{attribute 'GeneratedUsingTerminal: EL3413-0000-0019'}
{attribute addProperty BoxType "EL3413-0000-0019"}
{attribute addProperty Id "PM_Inputs_Channel_1AT %I*PM_Inputs_Channel_345EAE5425PM_Inputs_Channel_2AT %I*PM_Inputs_Channel_345EAE5425PM_Inputs_Channel_3AT %I*PM_Inputs_Channel_345EAE5425PM_Inputs_AuxiliaryAT %I*PM_Inputs_Auxiliary_3661DB6D9PM_Outputs_Channel_1AT %Q*PM_Outputs_Channel_E5FBDE301PM_Outputs_Channel_2AT %Q*PM_Outputs_Channel_E5FBDE301PM_Outputs_Channel_3AT %Q*PM_Outputs_Channel_E5FBDE301PM_Outputs_AuxiliaryAT %Q*PM_Outputs_Auxiliary_6BC1946F2WcStateAT %I*WcState_9091E0EB2InfoDataAT %I*InfoData_94A18F5E2"}
{attribute addProperty CRC "1122277636"}
{attribute addProperty Size "93"}
TYPE EL3413_42E49904 EXTENDS EtcSlaveTerminalBase_947E5A46 :
STRUCT
	{attribute addProperty Name "PM_Inputs_Channel_1"}
	PM_Inputs_Channel_1 : PM_Inputs_Channel_345EAE54;
	{attribute addProperty Name "PM_Inputs_Channel_2"}
	PM_Inputs_Channel_2 : PM_Inputs_Channel_345EAE54;
	{attribute addProperty Name "PM_Inputs_Channel_3"}
	PM_Inputs_Channel_3 : PM_Inputs_Channel_345EAE54;
	{attribute addProperty Name "PM_Inputs_Auxiliary"}
	PM_Inputs_Auxiliary : PM_Inputs_Auxiliary_3661DB6D;
	{attribute addProperty Name "PM_Outputs_Channel_1"}
	PM_Outputs_Channel_1 : PM_Outputs_Channel_E5FBDE30;
	{attribute addProperty Name "PM_Outputs_Channel_2"}
	PM_Outputs_Channel_2 : PM_Outputs_Channel_E5FBDE30;
	{attribute addProperty Name "PM_Outputs_Channel_3"}
	PM_Outputs_Channel_3 : PM_Outputs_Channel_E5FBDE30;
	{attribute addProperty Name "PM_Outputs_Auxiliary"}
	PM_Outputs_Auxiliary : PM_Outputs_Auxiliary_6BC1946F;
	{attribute addProperty Name "WcState"}
	WcState : WcState_9091E0EB;
	{attribute addProperty Name "InfoData"}
	InfoData : InfoData_94A18F5E;
END_STRUCT
END_TYPE

(* stored: Version 1.2.0.0, ProductVersion 3.1.4024.9
   DUT EL3413_42E49904: Id {908c176a-5aea-4312-983d-30292b4271fe} *)
